FUNCTION_BLOCK EL_LinearAxis (* LinearAxis: output values from its holder -> outputs (break before make); one holder at a time; all off on release or when the module aborts; inputs -> state channel when they change *)
  (* Standard: 61499-2 *)
  (* Version 0.1, 2026-09-28, Project contributors, AAU Smart Production Lab *)
  PACKAGE stoppering;
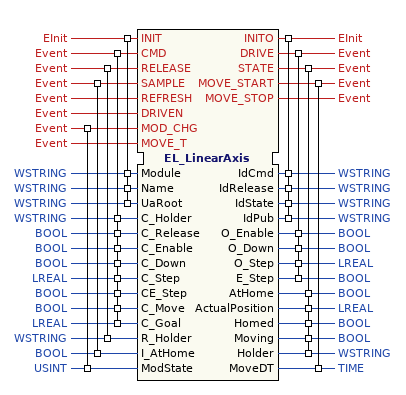
  EVENT_INPUT
    INIT : EInit WITH Module, Name, UaRoot;
    CMD WITH C_Holder, C_Release, C_Enable, C_Down, C_Step, CE_Step, C_Move, C_Goal;
    RELEASE WITH R_Holder;
    SAMPLE WITH I_AtHome;
    REFRESH;
    DRIVEN;
    MOD_CHG WITH ModState;
    MOVE_T;
  END_EVENT
  EVENT_OUTPUT
    INITO : EInit WITH IdCmd, IdRelease, IdState, IdPub;
    DRIVE WITH O_Enable, O_Down, O_Step, E_Step;
    STATE WITH AtHome, ActualPosition, Homed, Moving, Holder;
    MOVE_START WITH MoveDT;
    MOVE_STOP;
  END_EVENT
  VAR_INPUT
    Module : WSTRING;
    Name : WSTRING;
    UaRoot : WSTRING;
    C_Holder : WSTRING;
    C_Release : BOOL;
    C_Enable : BOOL;
    C_Down : BOOL;
    C_Step : LREAL;
    CE_Step : BOOL;
    C_Move : BOOL;
    C_Goal : LREAL;
    R_Holder : WSTRING;
    I_AtHome : BOOL;
    ModState : USINT;
  END_VAR
  VAR_OUTPUT
    IdCmd : WSTRING;
    IdRelease : WSTRING;
    IdState : WSTRING;
    IdPub : WSTRING;
    O_Enable : BOOL;
    O_Down : BOOL;
    O_Step : LREAL;
    E_Step : BOOL;
    AtHome : BOOL;
    ActualPosition : LREAL;
    Homed : BOOL;
    Moving : BOOL;
    Holder : WSTRING;
    MoveDT : TIME;
  END_VAR
  VAR
    Publish : BOOL;
    Beat : USINT;
    LastHolder : WSTRING;
    Pending : BOOL;
    OffPending : BOOL;
    L_AtHome : BOOL;
    L_Homed : BOOL;
    L_Moving : BOOL;
    N_Enable : BOOL;
    N_Down : BOOL;
    N_Step : LREAL;
    NE_Step : BOOL;
    N_Move : BOOL;
    N_Goal : LREAL;
    MoveGoal : LREAL;
    MoveFrom : LREAL;
    MoveDir : LREAL;
    MoveSince : TIME;
    MoveStart : BOOL;
    Uncounted : BOOL;
  END_VAR
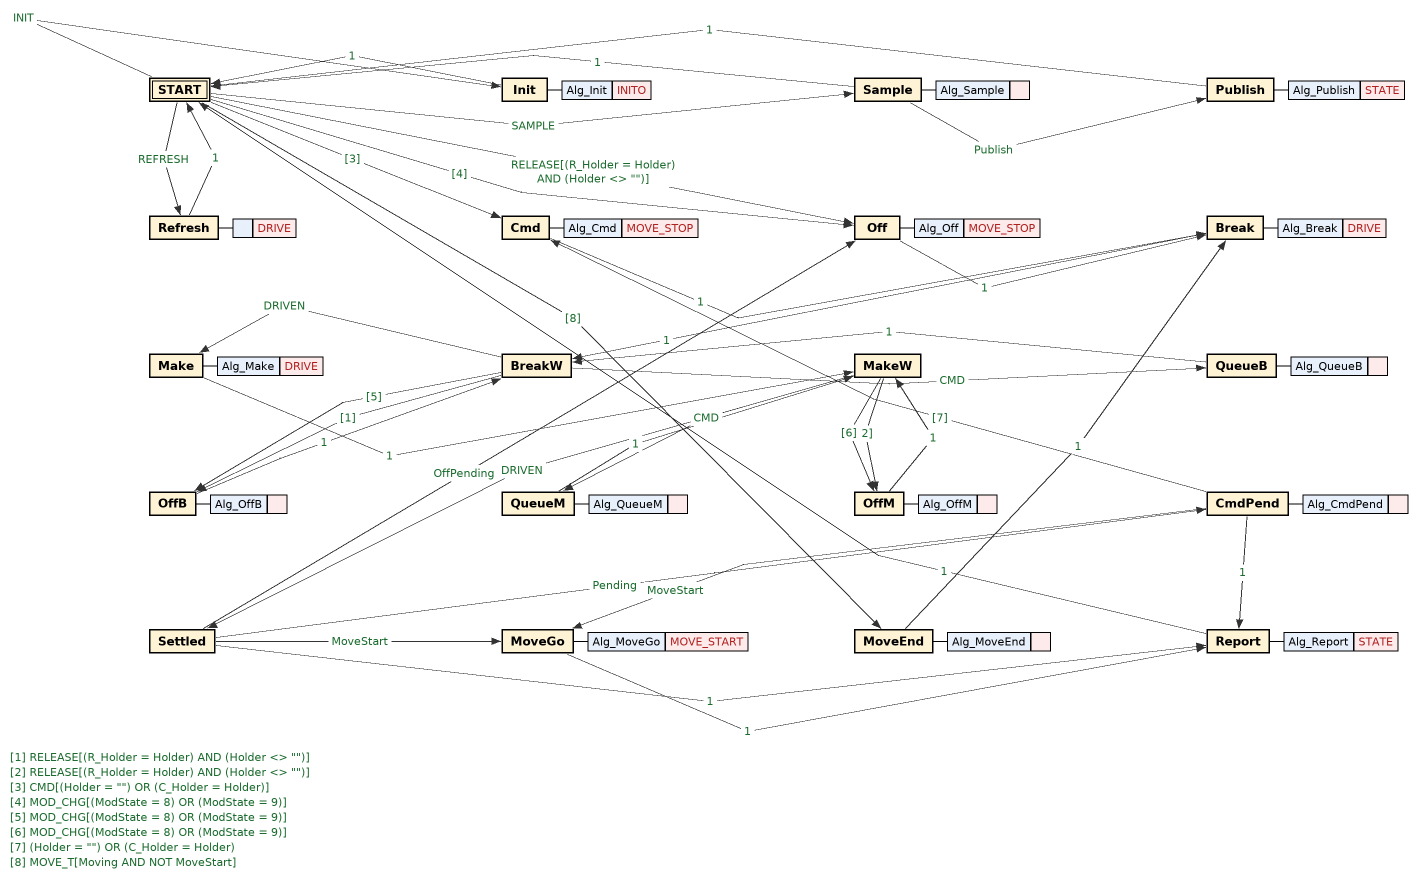
  EC_STATES
    START;
    Init : Alg_Init -> INITO;
    Sample : Alg_Sample;
    Publish : Alg_Publish -> STATE;
    Refresh : -> DRIVE;
    Cmd : Alg_Cmd -> MOVE_STOP;
    Off : Alg_Off -> MOVE_STOP;
    Break : Alg_Break -> DRIVE;
    Make : Alg_Make -> DRIVE;
    BreakW;
    MakeW;
    QueueB : Alg_QueueB;
    OffB : Alg_OffB;
    QueueM : Alg_QueueM;
    OffM : Alg_OffM;
    CmdPend : Alg_CmdPend;
    Settled;
    MoveGo : Alg_MoveGo -> MOVE_START;
    MoveEnd : Alg_MoveEnd;
    Report : Alg_Report -> STATE;
  END_STATES
  EC_TRANSITIONS
    START TO Init := INIT;
    START TO Sample := SAMPLE;
    START TO Refresh := REFRESH;
    START TO Cmd := CMD[(Holder = "") OR (C_Holder = Holder)];
    START TO Off := RELEASE[(R_Holder = Holder) AND (Holder <> "")];
    START TO Off := MOD_CHG[(ModState = 8) OR (ModState = 9)];
    START TO MoveEnd := MOVE_T[Moving AND NOT MoveStart];
    MoveEnd TO Break := 1;
    Init TO START := 1;
    Sample TO Publish := Publish;
    Sample TO START := 1;
    Publish TO START := 1;
    Refresh TO START := 1;
    Cmd TO Break := 1;
    Off TO Break := 1;
    Break TO BreakW := 1;
    BreakW TO Make := DRIVEN;
    Make TO MakeW := 1;
    MakeW TO Settled := DRIVEN;
    BreakW TO QueueB := CMD;
    BreakW TO OffB := RELEASE[(R_Holder = Holder) AND (Holder <> "")];
    BreakW TO OffB := MOD_CHG[(ModState = 8) OR (ModState = 9)];
    QueueB TO BreakW := 1;
    OffB TO BreakW := 1;
    MakeW TO QueueM := CMD;
    MakeW TO OffM := RELEASE[(R_Holder = Holder) AND (Holder <> "")];
    MakeW TO OffM := MOD_CHG[(ModState = 8) OR (ModState = 9)];
    QueueM TO MakeW := 1;
    OffM TO MakeW := 1;
    Settled TO Off := OffPending;
    Settled TO CmdPend := Pending;
    CmdPend TO Cmd := (Holder = "") OR (C_Holder = Holder);
    CmdPend TO MoveGo := MoveStart;
    Settled TO MoveGo := MoveStart;
    MoveGo TO Report := 1;
    CmdPend TO Report := 1;
    Settled TO Report := 1;
    Report TO START := 1;
  END_TRANSITIONS
  ALGORITHM Alg_Init IN ST:
IdCmd := CONCAT(CONCAT(CONCAT(CONCAT("loc[", Module), "/"), Name), "/cmd]");
IdRelease := CONCAT(CONCAT(CONCAT(CONCAT("loc[", Module), "/"), Name), "/release]");
IdState := CONCAT(CONCAT(CONCAT(CONCAT("loc[", Module), "/"), Name), "/state]");
IdPub := CONCAT(CONCAT(CONCAT(CONCAT(CONCAT(CONCAT(CONCAT(CONCAT(CONCAT(CONCAT(CONCAT(CONCAT(CONCAT(CONCAT(CONCAT(CONCAT(CONCAT("opc_ua[WRITE;", UaRoot), "/Equipment/"), Name), "/AtHome;"), UaRoot), "/Equipment/"), Name), "/ActualPosition;"), UaRoot), "/Equipment/"), Name), "/Homed;"), UaRoot), "/Equipment/"), Name), "/Moving"), "]");
  END_ALGORITHM
  ALGORITHM Alg_Sample IN ST:
AtHome := I_AtHome;
IF Moving AND NOT MoveStart THEN
  ActualPosition := MoveFrom + MoveDir * 20.0 * TIME_IN_MS_TO_LREAL(NOW_MONOTONIC() - MoveSince) / 1000.0;
  IF MoveDir * (ActualPosition - MoveGoal) > 0.0 THEN
    ActualPosition := MoveGoal;
  END_IF;
ELSIF AtHome THEN
  ActualPosition := 0.0;
  Homed := TRUE;
ELSIF Uncounted THEN
  Homed := FALSE;
END_IF;
Publish := (AtHome <> L_AtHome) OR (Homed <> L_Homed) OR (Moving <> L_Moving) OR (Holder <> LastHolder) OR (Beat >= 20) OR (Moving AND (Beat >= 4));
Beat := Beat + 1;
  END_ALGORITHM
  ALGORITHM Alg_Publish IN ST:
L_AtHome := AtHome;
L_Homed := Homed;
L_Moving := Moving;
LastHolder := Holder;
Beat := 0;
  END_ALGORITHM
  ALGORITHM Alg_Cmd IN ST:
Holder := C_Holder;
N_Enable := C_Enable;
N_Down := C_Down;
N_Step := C_Step;
NE_Step := CE_Step;
N_Move := C_Move;
N_Goal := C_Goal;
IF Moving AND NOT MoveStart THEN
  ActualPosition := MoveFrom + MoveDir * 20.0 * TIME_IN_MS_TO_LREAL(NOW_MONOTONIC() - MoveSince) / 1000.0;
  IF MoveDir * (ActualPosition - MoveGoal) > 0.0 THEN
    ActualPosition := MoveGoal;
  END_IF;
END_IF;
Moving := FALSE;
MoveStart := FALSE;
IF N_Move THEN
  IF Homed AND (ABS(N_Goal - ActualPosition) >= 0.0005) THEN
    MoveGoal := N_Goal;
    MoveFrom := ActualPosition;
    MoveDT := MUL_TIME(T#1s, ABS(N_Goal - ActualPosition) / 20.0);
    IF N_Goal > ActualPosition THEN
      MoveDir := 1.0;
      N_Enable := TRUE;
      N_Down := TRUE;
      N_Step := 50.0;
      NE_Step := TRUE;
    ELSE
      MoveDir := -1.0;
      N_Enable := TRUE;
      N_Down := FALSE;
      N_Step := 50.0;
      NE_Step := TRUE;
    END_IF;
    Moving := TRUE;
    MoveStart := TRUE;
  ELSE
    N_Enable := FALSE;
    N_Down := FALSE;
    N_Step := 0.0;
    NE_Step := FALSE;
  END_IF;
  Uncounted := FALSE;
ELSE
  Uncounted := N_Enable OR N_Down OR NE_Step;
END_IF;
IF C_Release THEN
  Holder := "";
END_IF;
  END_ALGORITHM
  ALGORITHM Alg_Off IN ST:
N_Enable := FALSE;
N_Down := FALSE;
N_Step := 0.0;
NE_Step := FALSE;
N_Move := FALSE;
N_Goal := 0.0;
IF Moving AND NOT MoveStart THEN
  ActualPosition := MoveFrom + MoveDir * 20.0 * TIME_IN_MS_TO_LREAL(NOW_MONOTONIC() - MoveSince) / 1000.0;
  IF MoveDir * (ActualPosition - MoveGoal) > 0.0 THEN
    ActualPosition := MoveGoal;
  END_IF;
END_IF;
Moving := FALSE;
MoveStart := FALSE;
Uncounted := FALSE;
Holder := "";
OffPending := FALSE;
  END_ALGORITHM
  ALGORITHM Alg_Break IN ST:
O_Enable := O_Enable AND N_Enable;
O_Down := O_Down AND N_Down;
  END_ALGORITHM
  ALGORITHM Alg_Make IN ST:
O_Enable := N_Enable;
O_Down := N_Down;
O_Step := N_Step;
E_Step := NE_Step;
  END_ALGORITHM
  ALGORITHM Alg_QueueB IN ST:
Pending := TRUE;
  END_ALGORITHM
  ALGORITHM Alg_OffB IN ST:
OffPending := TRUE;
  END_ALGORITHM
  ALGORITHM Alg_QueueM IN ST:
Pending := TRUE;
  END_ALGORITHM
  ALGORITHM Alg_OffM IN ST:
OffPending := TRUE;
  END_ALGORITHM
  ALGORITHM Alg_CmdPend IN ST:
Pending := FALSE;
  END_ALGORITHM
  ALGORITHM Alg_MoveGo IN ST:
MoveStart := FALSE;
MoveSince := NOW_MONOTONIC();
  END_ALGORITHM
  ALGORITHM Alg_MoveEnd IN ST:
ActualPosition := MoveGoal;
Moving := FALSE;
N_Enable := FALSE;
N_Down := FALSE;
N_Step := 0.0;
NE_Step := FALSE;
  END_ALGORITHM
  ALGORITHM Alg_Report IN ST:
LastHolder := Holder;
Beat := 0;
  END_ALGORITHM
END_FUNCTION_BLOCK
